Fanuc KAREL source: kc00032.KL

-- PROVISIONAL review KL for V770-1; original PC SHA256 e11f8c547e06aa92c578fc550c47960fc5b3b221c1e2709258b8e52200571b9c
-- Incomplete behavior may be omitted. Consult companion uncertainty JSON. Do not deploy.
PROGRAM KC00032
%NOLOCKGROUP
BEGIN
  -- UNRESOLVED_PC offsets 5-55; opcodes 27,22,2A,22,22,22,22,22,22,27,9D,31
  -- UNRESOLVED_PC offsets 60-64; opcodes 7F
END KC00032
